Staubli VAL3: sychronMove.pgx

public program sychronMove()
  local bool l_bTemp
  local num l_nCount
  local joint l_jTemp1
  local num l_nTime
begin
  //  //this task is synchronous moving
  //  //  MoveTo.trsf=cad:pCad[0].trsf
  //  //  l_bTemp=pointToJoint(tTool,jConfig,MoveTo,l_jTemp1)
  //  //  movej(l_jTemp1,tTool,mNomSpeed)
  //  //  waitEndMove()
  //  //  jConfig=herej()
  //  call FC_InitMotion()
  //  l_nCount=0
  //  bSetIO=true
  //  //
  //  nsumtime=clock()
  //  for l_nCount=0 to size(cad:pCad)-1
  //    //
  //    l_nTime=clock()
  //    //
  //    MoveTo.trsf=cad:pCad[l_nCount].trsf
  //    l_bTemp=pointToJoint(tTool,jConfig,MoveTo,l_jTemp1)
  //    $movejSync(l_jTemp1)
  //    //$movejSync(cad:jJointRx[l_nCount])
  //    l_nTime=clock()-l_nTime
  //    if l_nTime>nTime
  //      nTime=l_nTime
  //      nTestNum=l_nCount
  //    endIf
  //    delay(0)
  //  endFor
  //  //
  //  bSetIO=false
  //  //io:socket="(RBSTOP)"
  //  call FC_EndMotion()
  //  nsumtime=clock()-nsumtime
  //  popUpMsg("move end!")
  //  bTest=true
end
